(* CODESYS project CommanderC200_AutoRun.project

Project tree, tasks and I/O mapping:
  Drive : Commander C200, Nidec Control Techniques, version 1.9.4.1
    application Application
      Task Configuration
        Freewheeling
      program Freewheeling [LD]
    <Empty>
  Advanced Link Editor
*)

// Drive/Application/Freewheeling
PROGRAM Freewheeling
VAR
	timerWrite: TIME;
	timerCurrent: TIME;
	timerTest: TIME := T#60000MS;
	tempOk: BOOL;
	m1: BOOL;
	Timer_1: TON;
	Timer_MS: DINT;
	Timer_MS2: DINT;
	Timer_S: DINT;
	TON_0: TON;
	timerTest_1: DINT;
	Timer_S1: DINT;
	T1: TON;
	T2: TON;
	T11: BOOL;
	T12: BOOL;
END_VAR
VAR // added by the converter: edge detectors and wires of the graphical bodies
    _w1, _w2 : BOOL;
END_VAR

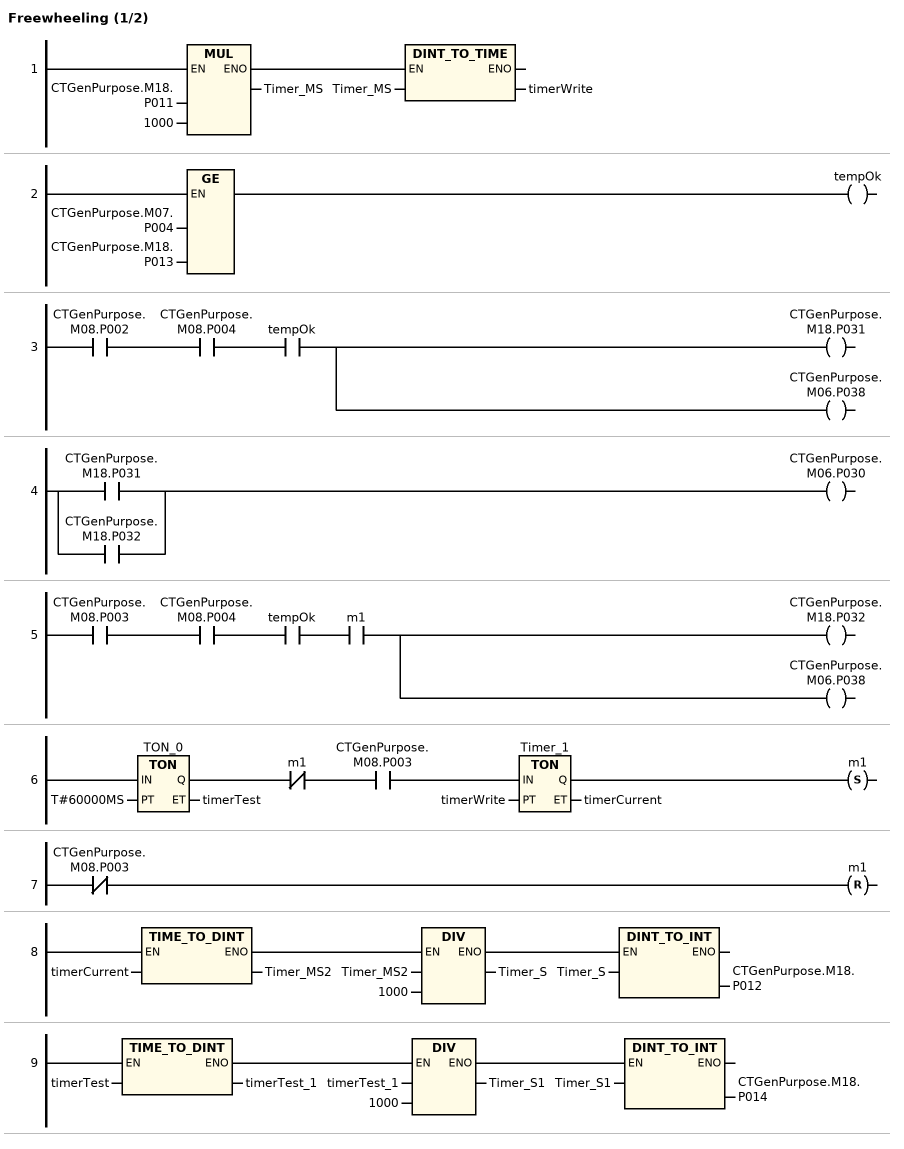
// NETWORK 1
Timer_MS := CTGenPurpose.M18.P011 * 1000;
timerWrite := DINT_TO_TIME(Timer_MS);

// NETWORK 2
tempOk := CTGenPurpose.M07.P004 >= CTGenPurpose.M18.P013;

// NETWORK 3
_w1 := CTGenPurpose.M08.P002 AND CTGenPurpose.M08.P004 AND tempOk;
CTGenPurpose.M18.P031 := _w1;
CTGenPurpose.M06.P038 := _w1;

// NETWORK 4
CTGenPurpose.M06.P030 := CTGenPurpose.M18.P031 OR CTGenPurpose.M18.P032;

// NETWORK 5
_w2 := CTGenPurpose.M08.P003 AND CTGenPurpose.M08.P004 AND tempOk AND m1;
CTGenPurpose.M18.P032 := _w2;
CTGenPurpose.M06.P038 := _w2;

// NETWORK 6
TON_0(IN := TRUE, PT := T#60000MS, ET => timerTest); // TON
Timer_1(IN := TON_0.Q AND NOT m1 AND CTGenPurpose.M08.P003, PT := timerWrite, ET => timerCurrent); // TON
m1 S= Timer_1.Q;

// NETWORK 7
m1 R= NOT CTGenPurpose.M08.P003;

// NETWORK 8
Timer_MS2 := TIME_TO_DINT(timerCurrent);
Timer_S := Timer_MS2 / 1000;
CTGenPurpose.M18.P012 := DINT_TO_INT(Timer_S);

// NETWORK 9
timerTest_1 := TIME_TO_DINT(timerTest);
Timer_S1 := timerTest_1 / 1000;
CTGenPurpose.M18.P014 := DINT_TO_INT(Timer_S1);

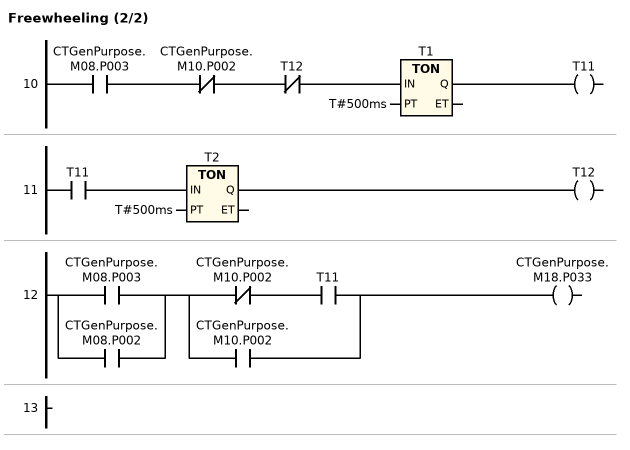
// NETWORK 10
T1(IN := CTGenPurpose.M08.P003 AND NOT CTGenPurpose.M10.P002 AND NOT T12, PT := T#500ms); // TON
T11 := T1.Q;

// NETWORK 11
T2(IN := T11, PT := T#500ms); // TON
T12 := T2.Q;

// NETWORK 12
CTGenPurpose.M18.P033 := (CTGenPurpose.M08.P003 OR CTGenPurpose.M08.P002) AND (NOT CTGenPurpose.M10.P002 AND T11 OR CTGenPurpose.M10.P002);

// NETWORK 13

END_PROGRAM
